// TwinCAT 3 PLC project PLC
// ProgramVersion: 3.1.4023.0
// libraries:
//   Tc2_EnOcean, * (Beckhoff Automation GmbH)
//   Tc2_Standard, * (Beckhoff Automation GmbH)
//   Tc2_System, * (Beckhoff Automation GmbH)
//   Tc3_Module, * (Beckhoff Automation GmbH)
// project tree:
//   / EnOceanCommunication.TcTTO, GlobalTextList.TcGTLO, PlcTask.TcTTO, Visualization Manager.TcVMO (not stored)
//   GVLs/ EnOcean.TcGVL, GUI.TcGVL, Hardware.TcGVL
//   POUs/ EnOceanCom.TcPOU, EnOceanSwitcher.TcPOU, MAIN.TcPOU, MotorControlProgram.TcPOU, ReceiveSwitch.TcPOU
//   VISUs/ Visualization.TcVIS
// real-time tasks:
//   TASK PlcTask: cycle T#10ms, priority 20, ADS port 350
//   TASK EnOceanCommunication: cycle T#5ms, priority 1, ADS port 351
// I/O:
//   DEVICE Device 1 (EtherCAT), AmsNetId 5.29.55.214.2.1
//     Term 1 (EK1100) [EK1100 EtherCAT Coupler (2A E-Bus)]
//       Term 2 (EL1008) [EL1008 8Ch. Dig. Input 24V, 3ms]
//       Term 3 (EL1008) [EL1008 8Ch. Dig. Input 24V, 3ms]
//       Term 4 (EL2008) [EL2008 8Ch. Dig. Output 24V, 0.5A]
//       Term 5 (EL2008) [EL2008 8Ch. Dig. Output 24V, 0.5A]
//       Term 6 (EL3002) [EL3002 2Ch. Ana. Input +/-10V]
//       Term 7 (EL4002) [EL4002 2Ch. Ana. Output 0-10V, 12bit]
//       Term 8 (EL3124) [EL3124 4Ch. Ana. Input 4-20mA Diff.]
//       Term 9 (EL4024) [EL4024 4Ch. Ana. Output 4-20mA, 12bit]
//       Box 10 (BK1250)
//     Term 11 (EK1100) [EK1100 EtherCAT Coupler (2A E-Bus)]
//       Term 12 (EL1819) [EL1819 16Ch. Dig. Input 24V, 10µs]
//       Term 13 (EL2008) [EL2008 8Ch. Dig. Output 24V, 0.5A]
//       Term 14 (EL4024) [EL4024 4Ch. Ana. Output 4-20mA, 12bit]
//       Term 15 (EL3024) [EL3024 4Ch. Ana. Input 4-20mA DIFF]
//       Term 16 (EL9011) [EL9011 End Terminal]
// variable links:
//   PLC/PLC Instance <-> Device 1 (EtherCAT)/Term 1 (EK1100)/Box 10 (BK1250)
//     EnOceanCommunication Inputs/EnOcean.stIn/CNODE <-> Term 2 (KL6581)/Channel 1/Input CNODE
//     EnOceanCommunication Inputs/EnOcean.stIn/DB{0..3} <-> Term 2 (KL6581)/Channel 1/Input DB{0..3}  (4 links)
//     EnOceanCommunication Inputs/EnOcean.stIn/ID{0..3} <-> Term 2 (KL6581)/Channel 1/Input ID{0..3}  (4 links)
//     EnOceanCommunication Inputs/EnOcean.stIn/ORG <-> Term 2 (KL6581)/Channel 1/Input ORG
//     EnOceanCommunication Inputs/EnOcean.stIn/STATUS <-> Term 2 (KL6581)/Channel 1/Input STATUS
//     EnOceanCommunication Inputs/EnOcean.stIn/nStatus <-> Term 2 (KL6581)/Channel 1/Status
//     EnOceanCommunication Outputs/EnOcean.stOut/CNODE <-> Term 2 (KL6581)/Channel 1/Output CNODE
//     EnOceanCommunication Outputs/EnOcean.stOut/DB{0..3} <-> Term 2 (KL6581)/Channel 1/Output DB{0..3}  (4 links)
//     EnOceanCommunication Outputs/EnOcean.stOut/ID{0..3} <-> Term 2 (KL6581)/Channel 1/Output ID{0..3}  (4 links)
//     EnOceanCommunication Outputs/EnOcean.stOut/ORG <-> Term 2 (KL6581)/Channel 1/Output ORG
//     EnOceanCommunication Outputs/EnOcean.stOut/STATUS <-> Term 2 (KL6581)/Channel 1/Output STATUS
//     EnOceanCommunication Outputs/EnOcean.stOut/nControl <-> Term 2 (KL6581)/Channel 1/Control
//   PLC/PLC Instance <-> Device 1 (EtherCAT)/Term 11 (EK1100)/Term 12 (EL1819)
//     PlcTask Inputs/Hardware.Motor1_Run_TAMU <-> Channel 3/Input
//     PlcTask Inputs/Hardware.Motor2_CircuitBreaker <-> Channel 1/Input
//     PlcTask Inputs/Hardware.Motor2_Error_TAMU <-> Channel 4/Input
//     PlcTask Inputs/Hardware.Motor2_Run_Contactor <-> Channel 2/Input
//   PLC/PLC Instance <-> Device 1 (EtherCAT)/Term 11 (EK1100)/Term 13 (EL2008)
//     PlcTask Outputs/Hardware.Motor1_Constant_speed <-> Channel 4/Output
//     PlcTask Outputs/Hardware.Motor1_Direction <-> Channel 3/Output
//     PlcTask Outputs/Hardware.Motor1_Start <-> Channel 2/Output
//     PlcTask Outputs/Hardware.Motor2_Start <-> Channel 1/Output
//   PLC/PLC Instance <-> Device 1 (EtherCAT)/Term 11 (EK1100)/Term 14 (EL4024)
//     PlcTask Outputs/Hardware.Motor1_speed_value <-> AO Outputs Channel 1/Analog output
//   PLC/PLC Instance <-> Device 1 (EtherCAT)/Term 11 (EK1100)/Term 15 (EL3024)
//     PlcTask Inputs/Hardware.Motor1_real_value <-> AI Standard Channel 1/Value

CONFIGURATION PLC
    RESOURCE PLC ON TwinCAT3
        TASK EnOceanCommunication(INTERVAL := T#5ms, PRIORITY := 1);
        TASK PlcTask(INTERVAL := T#10ms, PRIORITY := 20);
        PROGRAM EnOceanCom WITH EnOceanCommunication : EnOceanCom;
        PROGRAM MAIN WITH PlcTask : MAIN;
    END_RESOURCE
END_CONFIGURATION

// ---- GVLs/EnOcean.TcGVL
{attribute 'qualified_only'}
VAR_GLOBAL
	bInit: BOOL;
	nIndex: USINT;
	stIn  AT %I* : KL6581_Input;
	stOut AT %Q* : KL6581_Output;
	bComBusy: BOOL;
	bComError: BOOL;
	iCommErrorID: E_KL6581_Err;
	stBuffer: STR_KL6581;
	bComReady: BOOL;
	bStartSearch: BOOL;
	bSearchReceived: BOOL;
	iFoundDevice: INT;
	arrFoundIDs: ARRAY [0..255] OF DWORD;
	// switch
	stSwitchData: STR_EnOceanSwitch;
	bSwitchDataReceived: BOOL;
	dwSwitchID	:	DWORD := 16#FEFA6D21; 
	// sensor
	stThermoData: ARRAY [0..3] OF BYTE; // ST_EEP_A5_09_04;
	bThermoDataReceived: BOOL;
	dwThermoID	:	DWORD := 16#018DC339;
	
END_VAR

// ---- GVLs/GUI.TcGVL
{attribute 'qualified_only'}
VAR_GLOBAL
	//motors state
	bCMotor_Start		:BOOL;
	bVMotor_Start		:BOOL;
	bCMotor_Running		:BOOL;
	bVMotor_Running		:BOOL;
	bCMotor_Error		:BOOL;
	bVMotor_Error		:BOOL;
	//Variable motor
	iVMotor_CurrentSpeed	:INT;
	iVMotor_TargetSpeed		:INT;
	bVMotor_Direction		:BOOL; //directionof the motor, true left ---CHECK!!!!!
	bVMotor_ConstantSpeed	:BOOL;

END_VAR

// ---- GVLs/Hardware.TcGVL
{attribute 'qualified_only'}
VAR_GLOBAL
	Motor2_CircuitBreaker		AT %I*   : BOOL; //  1
	Motor2_Run_Contactor		AT %I*   : BOOL; //  2
	Motor1_Run_TAMU				AT %I*   : BOOL; //  3
	Motor2_Error_TAMU			AT %I*   : BOOL; //  4
	Motor2_Start				AT %Q*   : BOOL; //  1
	Motor1_Start				AT %Q*   : BOOL; //  2
	Motor1_Direction			AT %Q*   : BOOL; //  3
	Motor1_Constant_speed		AT %Q*   : BOOL; //  4
	Motor1_speed_value			AT %Q*   : INT; // Analog 1
	Motor1_real_value			AT %I*   : INT; // Analog 1
END_VAR

// ---- POUs/EnOceanCom.TcPOU
PROGRAM EnOceanCom
VAR
	fbKL6581: FB_KL6581;
	fbEnOceanSearch: FB_EnOcean_Search;
END_VAR

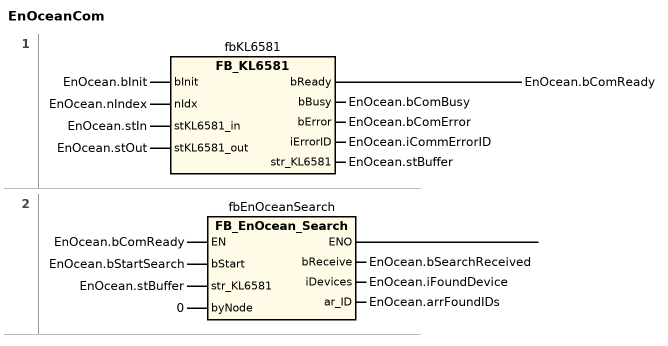
// NETWORK 1
fbKL6581(
    bInit := EnOcean.bInit,
    nIdx := EnOcean.nIndex,
    stKL6581_in := EnOcean.stIn,
    stKL6581_out := EnOcean.stOut,
    bBusy => EnOcean.bComBusy,
    bError => EnOcean.bComError,
    iErrorID => EnOcean.iCommErrorID,
    str_KL6581 => EnOcean.stBuffer); // FB_KL6581
EnOcean.bComReady := fbKL6581.bReady;

// NETWORK 2
IF EnOcean.bComReady THEN
    fbEnOceanSearch(
        bStart := EnOcean.bStartSearch,
        str_KL6581 := EnOcean.stBuffer,
        byNode := 0,
        bReceive => EnOcean.bSearchReceived,
        iDevices => EnOcean.iFoundDevice,
        ar_ID => EnOcean.arrFoundIDs); // FB_EnOcean_Search
END_IF

END_PROGRAM

// ---- POUs/MAIN.TcPOU
PROGRAM MAIN
VAR
END_VAR

MotorControlProgram();

END_PROGRAM

// ---- POUs/MotorControlProgram.TcPOU
PROGRAM MotorControlProgram
VAR
	rtCM_Start: R_TRIG;
	rtVM_Start: R_TRIG;
	rsCM	:	RS;
	rsVM	:	RS;
	
	targSpeed	:	INT;
END_VAR

(*
VAR_INPUT
	Run			:	BOOL;
	Direction	:	BOOL;
	ConstSpeed	:	BOOL;
	Velocity	:	INT;
END_VAR
VAR_OUTPUT
	isRunning	:	BOOL;
	iActualVel	:	INT;
END_VAR
*)



(* On / Off  Motor  *)

//***
rtCM_Start(CLK := GUI.bCMotor_Start);
rsCM(SET := rtCM_Start.Q);

Hardware.Motor2_Start := rsCM.Q1 ;


(*  TAMU  Motor  *)
//***
//rsVM(SET := GUI.bVMotor_Start);
//Hardware.Motor1_Start := rsVM.Q1 ;
Hardware.Motor1_Start :=  GUI.bVMotor_Start;
GUI.bVMotor_Running := Hardware.Motor1_Run_TAMU;
Hardware.Motor1_Constant_speed := GUI.bVMotor_ConstantSpeed;
Hardware.Motor1_Direction := GUI.bVMotor_Direction;
// Y = x0 + %% * Xrng
targSpeed := REAL_TO_INT( 32767 * (GUI.iVMotor_TargetSpeed / 100.0) );
Hardware.Motor1_speed_value := targSpeed;

GUI.iVMotor_CurrentSpeed := REAL_TO_INT( Hardware.Motor1_real_value / 32767.0 * 100.0 );

END_PROGRAM

// ---- POUs/EnOceanSwitcher.TcPOU
PROGRAM EnOceanSwitcher
VAR
	ftReceived: F_TRIG;
END_VAR

ftReceived(CLK:= EnOcean.bSwitchDataReceived, Q => received );
ftBtnBlue(CLK := GVL.btnBlue);

END_PROGRAM

// ---- POUs/ReceiveSwitch.TcPOU
PROGRAM ReceiveSwitch
VAR
	fbReceiveSwitchMessage: FB_Rec_RPS_Switch;
END_VAR

fbReceiveSwitchMessage(
	str_KL6581:= EnOcean.stBuffer, 
	byNode:= 0, 
	dw_ID:= EnOcean.dwSwitchID, 
	str_EnOceanSwitch=> EnOcean.stSwitchData, 
	by_Node=> , 
	bReceive=> EnOcean.bSwitchDataReceived);

END_PROGRAM

// ---- GlobalTextList.TcGTLO
TEXTLIST GlobalTextList
  889 = 'Constant Motor'
  67 = 'Constant speed'
  671 = 'Direction'
  890 = 'Error'
  86 = 'Running'
  279 = 'Variable Motor'
END_TEXTLIST

// ---- VISUs/Visualization.TcVIS
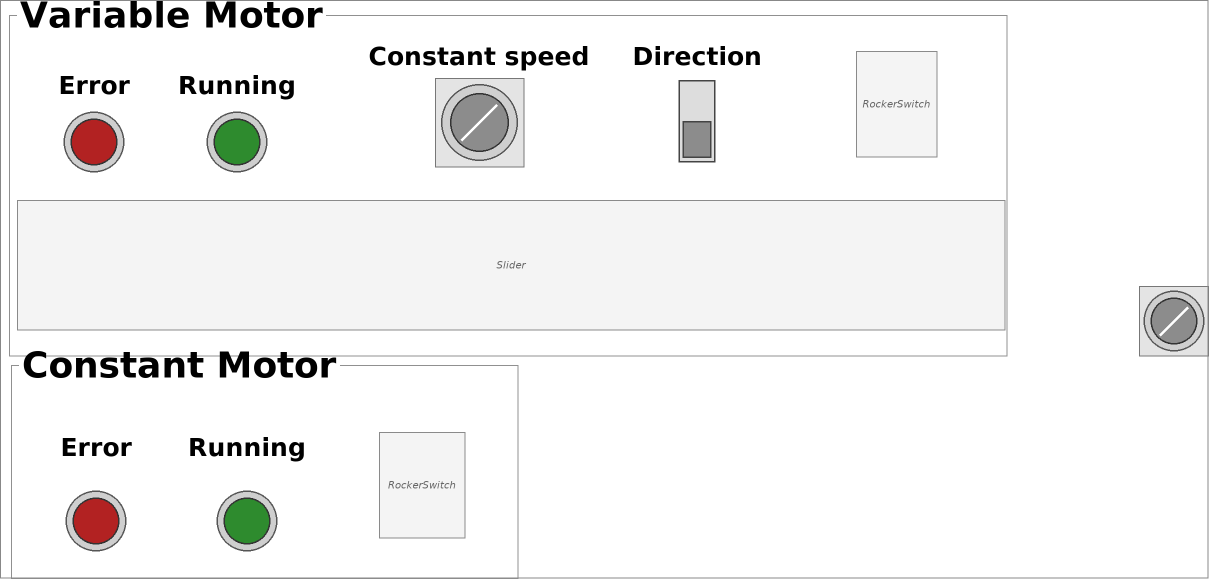
VISUALIZATION Visualization  // 1209x579
    Progressbar (40,261 940x19), variable: GUI.iVMotor_CurrentSpeed
    GroupBox (9,7 998x349), "Variable Motor"
        Lamp1 (50,100 70x70), variable: GUI.bVMotor_Error, style: Lamp-Lamp1-Red
        Label (325,16 290x66), "Constant speed"
        RotarySwitch (426,68 89x95), variable: GUI.bVMotor_ConstantSpeed, behaviour: TOGGLE, style: Switch-RotarySwitch-Gray
        Label (8,63 155x30), "Error"
        Lamp1 (193,100 70x70), variable: GUI.bVMotor_Running, style: Lamp-Lamp1-Green
        Label (163,425 150x30), "Running"
        RockerSwitch (847,44 81x106), variable: GUI.bVMotor_Start, behaviour: TOGGLE, style: Switch-RockerSwitch-Gray
        Slider (8,193 988x130), variable: GUI.iVMotor_TargetSpeed, scale 20..100
        DipSwitch (645,73 86x82), variable: GUI.bVMotor_Direction, behaviour: TOGGLE, style: Switch-DipSwitch-Gray
        Label (618,15 141x68), "Direction"
    Label (162,70 150x30), "Running"
    GroupBox (11,357 507x222), "Constant Motor"
        Lamp1 (50,129 70x70), variable: GUI.bCMotor_Error, style: Lamp-Lamp1-Red
        Label (752,84 216x30)
        Label (8,75 155x30), "Error"
        Lamp1 (201,129 70x70), variable: GUI.bCMotor_Running, style: Lamp-Lamp1-Green
        RockerSwitch (368,75 86x106), variable: GUI.bCMotor_Start, behaviour: TOGGLE, style: Switch-RockerSwitch-Gray
    RotarySwitch (1139,286 70x70), behaviour: TOGGLE, style: Switch-RotarySwitch-Gray
END_VISUALIZATION
